{attribute 'enable_dynamic_creation'}
FUNCTION_BLOCK RecipeStringValue IMPLEMENTS RecipeStringValueType
VAR
	_Name : T_MaxString;
	_Value : __SYSTEM.AnyType;
	_Assignment : STRING := ':=';
	_StringBoundary : STRING := '$'';
	
	sb : StringBuilderExtBuffer;
END_VAR

{attribute 'monitoring' := 'call'}
PROPERTY Assignment : STRING
GET
Assignment := _Assignment;
END_GET
SET
_Assignment := Assignment;
END_SET
END_PROPERTY

METHOD Bind
VAR_INPUT
	value : ANY;
END_VAR
_Value := value;
END_METHOD

PROPERTY Buffer : __SYSTEM.AnyType
GET
Buffer := sb.Buffer;
END_GET
SET
sb.Buffer := Buffer;
END_SET
END_PROPERTY

METHOD BuildAndGetAssignmentString : POINTER TO STRING
VAR_INPUT
END_VAR
sb.Clear();
sb.Append(
	BuildStringInline(_Name)
	.Append(' ')
	.Append(_Assignment)
	.Append(' ')
	.Append(_StringBoundary)
	.GetString()
);
sb.AppendByPointer(_Value.pValue);
sb.Append(_StringBoundary);
BuildAndGetAssignmentString := sb.BufferRef.pValue;
END_METHOD

METHOD Dispose
VAR_INPUT
END_VAR
__DELETE(THIS);
END_METHOD

{attribute 'monitoring' := 'call'}
PROPERTY Name : T_MaxString
GET
Name := _Name;
END_GET
SET
_Name := Name;
END_SET
END_PROPERTY

METHOD ParseAndAssignValue
VAR_INPUT
END_VAR
ClearDataAnyType(_Value);
MEMCPY(
	destAddr := _Value.pValue,
	srcAddr := sb.BufferRef.pValue,
	n := MIN(DINT_TO_UDINT(_Value.diSize - 1), LEN2(sb.BufferRef.pValue))
);
END_METHOD

{attribute 'monitoring' := 'call'}
PROPERTY ValueString : T_MaxString
GET
IF (IsAnyTypeBinded(_Value)) THEN
	ValueString := AnyTypeToString(_Value);
END_IF
END_GET
END_PROPERTY

END_FUNCTION_BLOCK

(* stored: Version 1.1.0.1, ProductVersion 3.1.4024.15
   POU RecipeStringValue: Id {43392db2-3186-0f20-0440-012ad562e1ba}, SpecialFunc None
   Property Assignment: Id {2806e733-14e8-0b63-24e2-541ced433e0c}
   Get Get: Id {bafcbdb4-2285-0133-2a2d-a43de1b22af5}
   Set Set: Id {82ded797-581e-0bb8-10f2-781d42f935ae}
   Method Bind: Id {951222a6-3de3-0ef0-3691-d46d19023f8b}
   Property Buffer: Id {a0a63aa0-e81a-097a-37c1-f9f141841650}
   Get Get: Id {0264b3de-f633-0087-0acc-47000fdd0dad}
   Set Set: Id {6e95e0f7-0f8b-02e4-19ca-17859d37edde}
   Method BuildAndGetAssignmentString: Id {52adad33-eaab-0122-1b47-ee42c7f83c26}
   Method Dispose: Id {bb685d27-573d-06ee-22f0-673d4b91a5e7}
   Property Name: Id {81d82b19-7c47-08a8-1737-8d4a4ebabf36}
   Get Get: Id {9599f689-243d-0fe0-25ba-9b2a71610801}
   Set Set: Id {08db63f8-ae4c-0185-0e00-fbdf30a1f508}
   Method ParseAndAssignValue: Id {427b66df-02cd-019e-2798-ca99d2de8b7e}
   Property ValueString: Id {56c8276b-9df7-0124-31aa-00ecd70e1926}
   Get Get: Id {c9d99e8d-b3b0-0707-1c78-97db7e41be46} *)
